(* IEC 61131-3 sources: volt/packages/volt-lsp-iec/test-corpus/lenze-mid/Device/Plc Logic/Application/Library Manager/L_OEEA_MachineDowntimeSolution, 3.26.4.8 (Lenze), 8 files *)

(* ---- EPRODUCTION_LOG.dut ---- *)
TYPE EPRODUCTION_LOG :
(
	TEXT := 0,
	JSON := 1
);
END_TYPE

(* ---- UERRORNUMBER.dut ---- *)
TYPE UERRORNUMBER :
UNION
	DWERRORNUMBER : DWORD;
	AWERRORINFO : ARRAY [1..2] OF WORD;
END_UNION
END_TYPE

(* ---- VERSIONCONSTANTS.gvl ---- *)
VAR_GLOBAL
	GC_BYAMOUNTOFGENERALDATA : BYTE := 50;
	GC_BYAMOUNTDOWNTIMEERRORS : BYTE := 10;
	GC_IFILTERSAMPLES : INT := 20;
END_VAR

(* ---- L_DOWNTIME_BASE.pou ---- *)
FUNCTION_BLOCK L_DOWNTIME_BASE
VAR_INPUT
	XENABLE : BOOL;
	XACTIVATELOG : BOOL;
	XRESETLOG : BOOL;
	XRESETPRODLOG : BOOL;
	XUSERESONCODESTRING : BOOL;
	SRESONCODESTRING : STRING;
END_VAR
VAR_IN_OUT
	SCSHIFTVALUES : scCurrentShiftValues;
	SCPDINTERNAL : scInternalDownVar;
END_VAR
VAR
	SCCLEARLOGVALUES : scDowntime_base;
	SDATETIMEDIFF : STRING;
	SDATETIME : STRING;
	SCUTTIMESTR : STRING;
	IPRODUCTIONMODE : INT;
	TDATETIMEDIFF : TIME;
	XFIRSTCYCLE : BOOL;
END_VAR
END_FUNCTION_BLOCK

METHOD ACT_INCREMENT_LOG : BOOL
VAR_IN_OUT
	SCSHIFTVALUES : scCurrentShiftValues;
	SCPDINTERNAL : scInternalDownVar;
END_VAR
END_METHOD

METHOD ACT_STOREPD_BASE : BOOL
VAR_IN_OUT
	SCMACHINEDATA : scMachineData_base;
	SCPDINTERNAL : scInternalDownVar;
END_VAR
END_METHOD

METHOD ACT_DOWNTIME_SUB_LOGBOOK_JSON : BOOL
VAR_INPUT
	STYPE : STRING;
END_VAR
VAR_IN_OUT
	SCMACHINEDATA : scMachineData_base;
	SCDOWNTIME : scDowntime_base;
	SCSHIFTVALUES : scCurrentShiftValues;
	SCPDINTERNAL : scInternalDownVar;
END_VAR
END_METHOD

METHOD ACT_MAIN_BASE : BOOL
VAR_IN_OUT
	SCMACHINEDATA : scMachineData_base;
	SCDOWNTIME : scDowntime_base;
	SCSHIFTVALUES : scCurrentShiftValues;
	SCPDINTERNAL : scInternalDownVar;
END_VAR
END_METHOD

METHOD ACT_DOWNTIME_BASE_LOGBOOK : BOOL
VAR_IN_OUT
	SCMACHINEDATA : scMachineData_base;
	SCDOWNTIME : scDowntime_base;
	SCSHIFTVALUES : scCurrentShiftValues;
	SCPDINTERNAL : scInternalDownVar;
END_VAR
END_METHOD

METHOD ACT_DOWNTIME_SUB_LOGBOOK_JSON_DURATION : BOOL
VAR_IN_OUT
	SCDOWNTIME : scDowntime_base;
	SCSHIFTVALUES : scCurrentShiftValues;
	SCPDINTERNAL : scInternalDownVar;
END_VAR
END_METHOD

(* ---- L_OEEA_DOWNTIME.pou ---- *)
FUNCTION_BLOCK L_OEEA_DOWNTIME EXTENDS L_Downtime_base
VAR_INPUT
	EPRODLOGFORMAT : eProduction_log;
END_VAR
VAR_OUTPUT
	SCACTUALSTATEDURATION : scVisuProductionStatus_base;
END_VAR
VAR_IN_OUT
	SCMACHINEDATA : scMachineData;
	SCDOWNTIME : scDowntime;
END_VAR
VAR
	XLOGRECORDING : BOOL;
	XLOGRECORDING2 : BOOL;
	SCLEARRESULTLOG : scDowntime_Log;
	IPOSSTR : INT;
	IPOSSTR2 : INT;
	ILENGHT : INT;
	SCSHIFTCHANGEDOWNTIME : scDowntime;
	SRESULT : STRING(255);
	SRESULT2 : STRING(255);
	STYPE : STRING;
	I : INT;
	J : INT;
	K : INT;
	L : INT;
	IINDEX : ARRAY [1..3] OF INT;
	IINDEXCLEAR : ARRAY [1..3] OF INT;
	IINDEX2 : ARRAY [1..3] OF INT;
	IINDEX3 : ARRAY [1..3] OF INT;
	DIDURATION : ARRAY [1..3] OF DINT;
	DIDURATIONCLEAR : ARRAY [1..3] OF DINT;
	DIDURATION2 : ARRAY [1..3] OF DINT;
	DIDURATION3 : ARRAY [1..3] OF DINT;
	DTLASTCURRENTTIME : TIME_OF_DAY;
END_VAR
END_FUNCTION_BLOCK

METHOD ACT_TOP3
END_METHOD

METHOD ACT_DOWNTIMESTATISTIC
END_METHOD

METHOD ACT_SHIFTEVENT
END_METHOD

METHOD ACT_SHIFTDATA
END_METHOD

METHOD ACT_DOWNTIME_LOGBOOK
END_METHOD

METHOD ACT_DOWNTIME_SUB_LOGBOOK_TEXT
END_METHOD

METHOD ACT_STATEDURATION
END_METHOD

(* ---- L_OEEA_DOWNTIME_BASE.pou ---- *)
FUNCTION_BLOCK L_OEEA_DOWNTIME_BASE EXTENDS L_Downtime_base
VAR_IN_OUT
	SCMACHINEDATA : scMachineData_base;
	SCDOWNTIME : scDowntime_base;
END_VAR
VAR
	XLOGRECORDING : BOOL;
	XLOGRECORDING2 : BOOL;
	SCSHIFTCHANGEDOWNTIME : scDowntime_base;
END_VAR
END_FUNCTION_BLOCK

METHOD ACT_SHIFTEVENT
END_METHOD

(* ---- L_OEEA_SHIFTDOWNTIMEHISTORY.pou ---- *)
FUNCTION_BLOCK L_OEEA_SHIFTDOWNTIMEHISTORY
VAR_INPUT
	XENABLE : BOOL;
	XRESETHISTORY : BOOL;
END_VAR
VAR_IN_OUT
	SCSHIFTDOWNTIME : scDowntime;
	SCSHIFTVALUES : scCurrentShiftValues;
	SCSHIFTDOWNTIMEHISTORY : ARRAY [1..3] OF scDowntime;
END_VAR
VAR
	SCSHIFTCHANGEDOWNTIME : scDowntime;
	I : INT;
	ISHFTCHANGECOUNTER : INT;
END_VAR
END_FUNCTION_BLOCK

(* ---- L_OEEA_SHIFTDOWNTIMEHISTORY_BASE.pou ---- *)
FUNCTION_BLOCK L_OEEA_SHIFTDOWNTIMEHISTORY_BASE
VAR_INPUT
	XENABLE : BOOL;
	XRESETHISTORY : BOOL;
END_VAR
VAR_IN_OUT
	SCSHIFTDOWNTIME : scDowntime_base;
	SCSHIFTVALUES : scCurrentShiftValues;
	SCSHIFTDOWNTIMEHISTORY : ARRAY [1..3] OF scDowntime_base;
END_VAR
VAR
	SCSHIFTCHANGEDOWNTIME : scDowntime;
	I : INT;
	ISHFTCHANGECOUNTER : INT;
END_VAR
END_FUNCTION_BLOCK
